(* PLC project v0.6.02_RefactorGateAndTest.project, CODESYS CODESYS V3.5 SP19 Patch 1 *)
(* stored: creationDateTime 2026-08-14T10:10:49.359610, modificationDateTime 2026-08-14T10:10:49.359610 *)

(* ═══════════════════════════════════════════════════════════════ 🔧 ST_DredgingAssistCfg — Réglages persistants assistants prélèvement 📄 Doc : DOC/AF/AF_Partie-04_Mode_SemiAuto_Sequenceur_v2.0.md §3ter ═══════════════════════════════════════════════════════════════ *)
TYPE ST_DredgingAssistCfg : STRUCT
  DiveStartMin_M : REAL := 1;  (* Position mini M1/M2 avant plongée *)
  ImmersionUpper_M : REAL := 0.5;  (* Borne haute fenêtre front immersion *)
  ImmersionLower_M : REAL := -0.5;  (* Borne basse fenêtre front immersion *)
  ExtractionControlDistance_M : REAL := 2;  (* Remontée palier 1 avant accélération *)
  TglEnableDiveSearch : BOOL := TRUE;  (* Mode assistance plongée mémorisé *)
  TglEnableExtractionSequence : BOOL := TRUE;  (* Mode assistance extraction mémorisé *)
  TglEnableDumpAtTremie : BOOL := TRUE;  (* Mode assistance vidage trémie mémorisé *)
  Initialized : BOOL := FALSE;  (* Pont persistance/IHM initialisé *)
END_STRUCT;
END_TYPE

(* ═══════════════════════════════════════════════════════════════ 🌉 FB_CfgPersistBridge_DredgingAssistCfg — Pont IHM/persistance prélèvement ═══════════════════════════════════════════════════════════════ *)
FUNCTION_BLOCK FB_CfgPersistBridge_DredgingAssistCfg
  VAR_OUTPUT
    JustRestored : BOOL;
  END_VAR
  VAR_IN_OUT
    Hmi : ST_DredgingAssistCfg;
    Persist : ST_DredgingAssistCfg;
  END_VAR

            

JustRestored := FALSE;
IF NOT Hmi.Initialized THEN
    Hmi := Persist;
    Hmi.Initialized := TRUE;
    JustRestored := TRUE;
ELSE
    Persist := Hmi;
END_IF;

          
END_FUNCTION_BLOCK
